FUNCTION_BLOCK AnalogInput_1
VAR
	nMaxRawValue: REAL := 7812500;  // for 24 bit device, e.g. ELM300x - check manual
	nRawValue AT %I*: DINT; // signed 32 bit integer representing full value range
	fMaxVoltage: REAL := 10; // measurement range
	valuebuffer: CounterTimer; // buffer for timed measurements
	filterbuffer: FilterRingBuffer;
	nFilterSize: UDINT := 100;
	fVoltage: REAL;
	fVoltageFiltered: REAL; // running average filter
END_VAR

fVoltage := fMaxVoltage * DINT_TO_REAL(nRawValue) / nMaxRawValue;  

IF filterbuffer.nBufferSize <> nFilterSize THEN
	nFilterSize := filterbuffer.SetFilterSize(nFilterSize);
END_IF
filterbuffer.Store(fVoltage);
fVoltageFiltered := filterbuffer.CalculateMean();

valuebuffer(fValue:=fVoltage);  // makes sure buffer in initialized and calls StoreValueConditional

END_FUNCTION_BLOCK

(* stored: Version 1.1.0.1, ProductVersion 3.1.4024.12
   POU AnalogInput_1: Id {e4609ea9-c11a-429c-aa7a-7ca0edc7ff9d}, SpecialFunc None *)
